// TwinCAT 3 PLC project TestCode
// ProgramVersion: 3.1.4022.3
// libraries:
//   Tc2_Standard, * (Beckhoff Automation GmbH)
//   Tc2_System, * (Beckhoff Automation GmbH)
//   Tc3_Module, * (Beckhoff Automation GmbH)
// project tree:
//   GVLs/ DUT.TcTLEO (not stored), VARS.TcGVL (not stored)
//   / PlcTask.TcTTO
//   POUs/ MAIN.TcPOU

CONFIGURATION TestCode
    RESOURCE PLC ON TwinCAT3
        TASK PlcTask(INTERVAL := T#10ms, PRIORITY := 4);
        PROGRAM MAIN WITH PlcTask : MAIN;
    END_RESOURCE
END_CONFIGURATION

// ---- POUs/MAIN.TcPOU
PROGRAM MAIN
VAR
	heartbeat : BYTE;
	out1 AT %Q* : BOOL;
	outVal1 : BOOL;
END_VAR

VARS.iSum := VARS.iTest1 + VARS.iTest2;
//heartbeat:= heartbeat+1;
out1 := outval1;
VARS.eTestEnumRbv := VARS.eTestEnum;

END_PROGRAM
